// TwinCAT 3 PLC project testStepper
// ProgramVersion: 3.1.4023.0
// libraries:
//   Tc2_MC2, * (Beckhoff Automation GmbH)
//   Tc2_NC, * (Beckhoff Automation GmbH)
//   Tc2_Standard, * (Beckhoff Automation GmbH)
//   Tc2_System, * (Beckhoff Automation GmbH)
//   Tc3_Module, * (Beckhoff Automation GmbH)
//   VisuDialogs, * (System)
// project tree:
//   / GlobalTextList.TcGTLO (not stored), PlcTask.TcTTO (not stored), Visualization Manager.TcVMO (not stored)
//   GVLs/ GVL_AxisCtr.TcGVL (not stored), GVL_IO.TcGVL (not stored), GVL_NC.TcGVL (not stored)
//   POUs/ Command_to_Action.TcPOU, DegreesToRelativeMovment.TcPOU (not stored), movements.TcPOU, PositionToDegree.TcPOU (not stored), MAIN.TcPOU, POUNCPowerOn.TcPOU (not stored)
//   VISUs/ testStepperVisu.TcVIS

// ---- POUs/Command_to_Action.TcPOU
FUNCTION_BLOCK Command_to_Action
VAR_INPUT
	inputString : STRING;
END_VAR
VAR_OUTPUT
	recognitionValue : REAL;
END_VAR
VAR
	putString : STRING;
	recognitionString : STRING := 'Steer(';
	stringLength : int;
END_VAR

IF FIND(STR1:= inputString  , STR2:= recognitionString ) = 1 THEN
	putString := DELETE(STR:=inputString , LEN:= 6 , POS:=1 );
	stringLength := LEN(putstring);
	putString := DELETE(STR:=putString , LEN:= 1 , POS:= stringLength);
	recognitionValue := STRING_TO_INT(putString);
END_IF

END_FUNCTION_BLOCK

// ---- POUs/movements.TcPOU
PROGRAM movements
VAR
	MC_MoveAbsolute_0: MC_MoveAbsolute;
	ExecuteMovement : BOOL;
	
	movementBuffer : MC_BufferMode; 
	
	DegreesToRelativeMovment_0: DegreesToRelativeMovment;
	
	Command_to_Action_0: Command_to_Action;
	
	PositionToDegree_0: PositionToDegree;
END_VAR

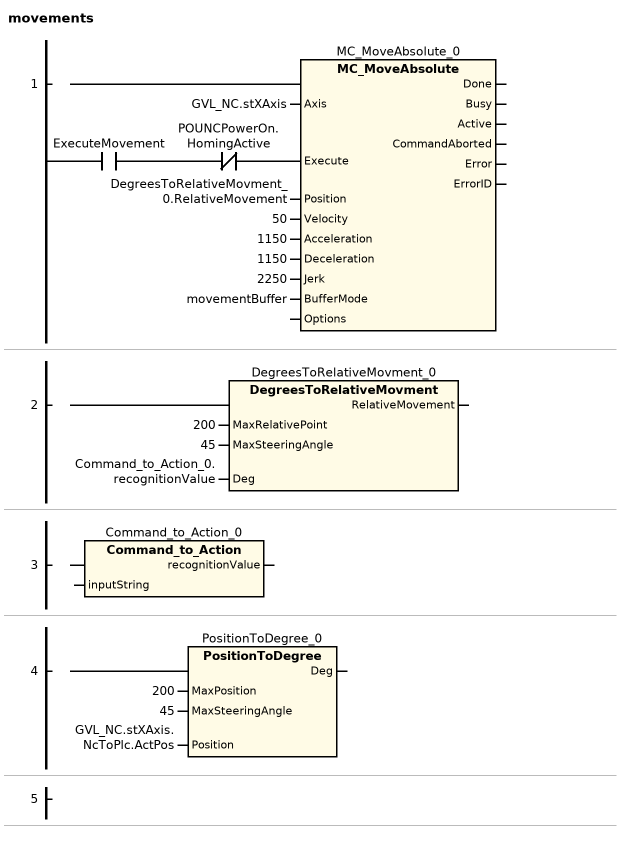
// NETWORK 1
MC_MoveAbsolute_0(
    Axis := GVL_NC.stXAxis,
    Execute := ExecuteMovement AND NOT POUNCPowerOn.HomingActive,
    Position := DegreesToRelativeMovment_0.RelativeMovement,
    Velocity := 50,
    Acceleration := 1150,
    Deceleration := 1150,
    Jerk := 2250,
    BufferMode := movementBuffer); // MC_MoveAbsolute

// NETWORK 2
DegreesToRelativeMovment_0(
    MaxRelativePoint := 200,
    MaxSteeringAngle := 45,
    Deg := Command_to_Action_0.recognitionValue); // DegreesToRelativeMovment

// NETWORK 3
Command_to_Action_0(); // Command_to_Action

// NETWORK 4
PositionToDegree_0(MaxPosition := 200, MaxSteeringAngle := 45, Position := GVL_NC.stXAxis.NcToPlc.ActPos); // PositionToDegree

// NETWORK 5

END_PROGRAM

// ---- POUs/MAIN.TcPOU
PROGRAM MAIN
VAR
	fbReadXaxisStatus: MC_ReadStatus;
	
END_VAR

fbReadXaxisStatus(
	Axis:=GVL_NC.stXAxis , 
	Enable:= GVL_AxisCtr.bXAxisEnable , 
	Valid=> , 
	Busy=> , 
	Error=> , 
	ErrorID=> , 
	ErrorStop=> , 
	Disabled=> , 
	Stopping=> , 
	StandStill=> , 
	DiscreteMotion=> , 
	ContinuousMotion=> , 
	SynchronizedMotion=> , 
	Homing=> , 
	ConstantVelocity=> , 
	Accelerating=> , 
	Decelerating=> , 
	Status=> GVL_NC.stXaxisStatus);
	POUNCPowerOn();
	movements();

END_PROGRAM

// ---- VISUs/testStepperVisu.TcVIS
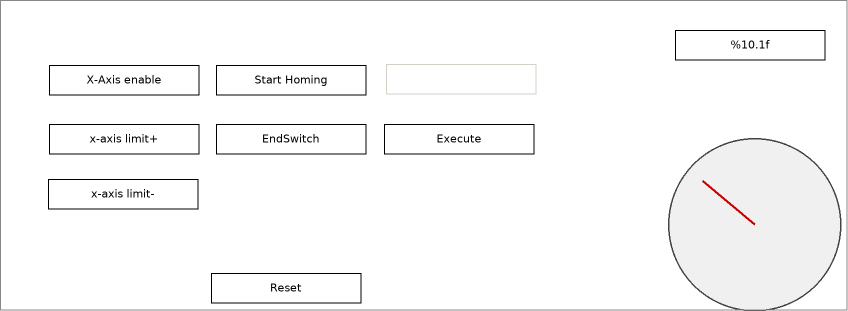
VISUALIZATION testStepperVisu  // 848x311
    Rectangle (49,65 150x30), "X-Axis enable"
        toggle GVL_AxisCtr.bXAxisEnable
    RoundedRectangle (49,124 150x30), "x-axis limit+", colour toggle: GVL_IO.I_bXAxisLimitSwPos
        toggle GVL_IO.I_bXAxisLimitSwPos
    RoundedRectangle (48,179 150x30), "x-axis limit-", colour toggle: GVL_IO.I_bXAxisLimitSwNeg
        toggle GVL_IO.I_bXAxisLimitSwNeg
    Rectangle (675,30 150x30), "%10.1f", text variable: GVL_NC.stXAxis.NcToPlc.ActPos
    Rectangle (384,124 150x30), "Execute"
        tap movements.ExecuteMovement
    Rectangle (216,65 150x30), "Start Homing"
        tap POUNCPowerOn.StartHoming
    Rectangle (216,124 150x30), "EndSwitch"
        toggle POUNCPowerOn.endSW
    Rectangle (211,273 150x30), "Reset"
        tap POUNCPowerOn.reset
    Meter90 (661,138 187x173), value: movements.PositionToDegree_0.Deg, style: Meter-Meter90-Gray, scale format: %.1f, scale -45..45
    Textfield (386,64 150x30), text variable: movements.Command_to_Action_0.inputString
        OnMouseDown: write the text variable via Default
END_VISUALIZATION
